TYPE ST_RepetitionRate :
STRUCT
	RepRateAboveThresholdSt : BOOL;
	RepetitionRateHzSt : REAL;
	RepetitionRateHzThreshold : REAL;
END_STRUCT
END_TYPE

(* stored: Version 1.1.0.1, ProductVersion 3.1.4024.5
   DUT ST_RepetitionRate: Id {3e1b9375-10c8-4393-b377-563ae32a885a} *)
